// Mitsubishi GX Works2 project: PLC 특수기능 (신호의 펄스화)   PLC: Q03UDV

PROGRAM MAIN
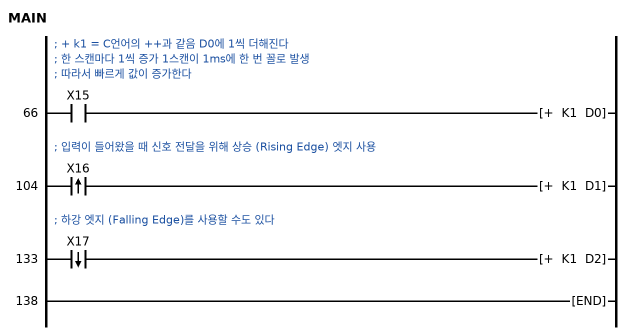
; + k1 = C언어의 ++과 같음 D0에 1씩 더해진다
; 한 스캔마다 1씩 증가 1스캔이 1ms에 한 번 꼴로 발생
; 따라서 빠르게 값이 증가한다
66    LD      X15
      +       K1 D0
; 입력이 들어왔을 때 신호 전달을 위해 상승 (Rising Edge) 엣지 사용
104   LDP     X16
      +       K1 D1
; 하강 엣지 (Falling Edge)를 사용할 수도 있다
133   LDF     X17
      +       K1 D2
138   END
END_PROGRAM
